FUNCTION_BLOCK FB_LoopController
VAR_INPUT
END_VAR
VAR_OUTPUT
END_VAR
VAR
END_VAR

END_FUNCTION_BLOCK

(* stored: Version 1.1.0.1, ProductVersion 3.1.4024.16
   POU FB_LoopController: Id {f48adaf0-df81-44d4-869d-09b0da41d4aa}, SpecialFunc None *)
